# EPICS autosave request: leybold/read_write_int_floatE_settings.req
$(P):$(FPARAM)
$(P):$(IPARAM)
